FUNCTION_BLOCK FiveStateActuator (* Basic Function Block Type *)
  (* Standard: 61499-2 *)
  (* Version 0.0, 5/13/2025, azam_w, Schneider Electric, Template *)
  PACKAGE Main;
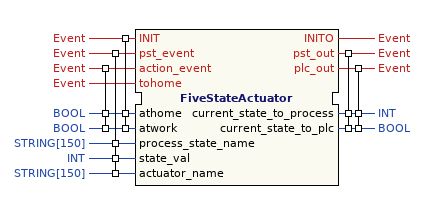
  EVENT_INPUT
    INIT WITH athome, atwork;
    pst_event WITH process_state_name, state_val, actuator_name; (* Normal Execution Request *)
    action_event WITH athome, atwork;
    tohome;
  END_EVENT
  EVENT_OUTPUT
    INITO;
    pst_out WITH current_state_to_process, current_state_to_plc; (* Execution Confirmation *)
    plc_out WITH current_state_to_plc, current_state_to_process;
  END_EVENT
  VAR_INPUT
    athome : BOOL;
    atwork : BOOL;
    process_state_name : STRING[150];
    state_val : INT;
    actuator_name : STRING[150];
  END_VAR
  VAR_OUTPUT
    current_state_to_process : INT; (* Output event qualifier *)
    current_state_to_plc : BOOL;
  END_VAR
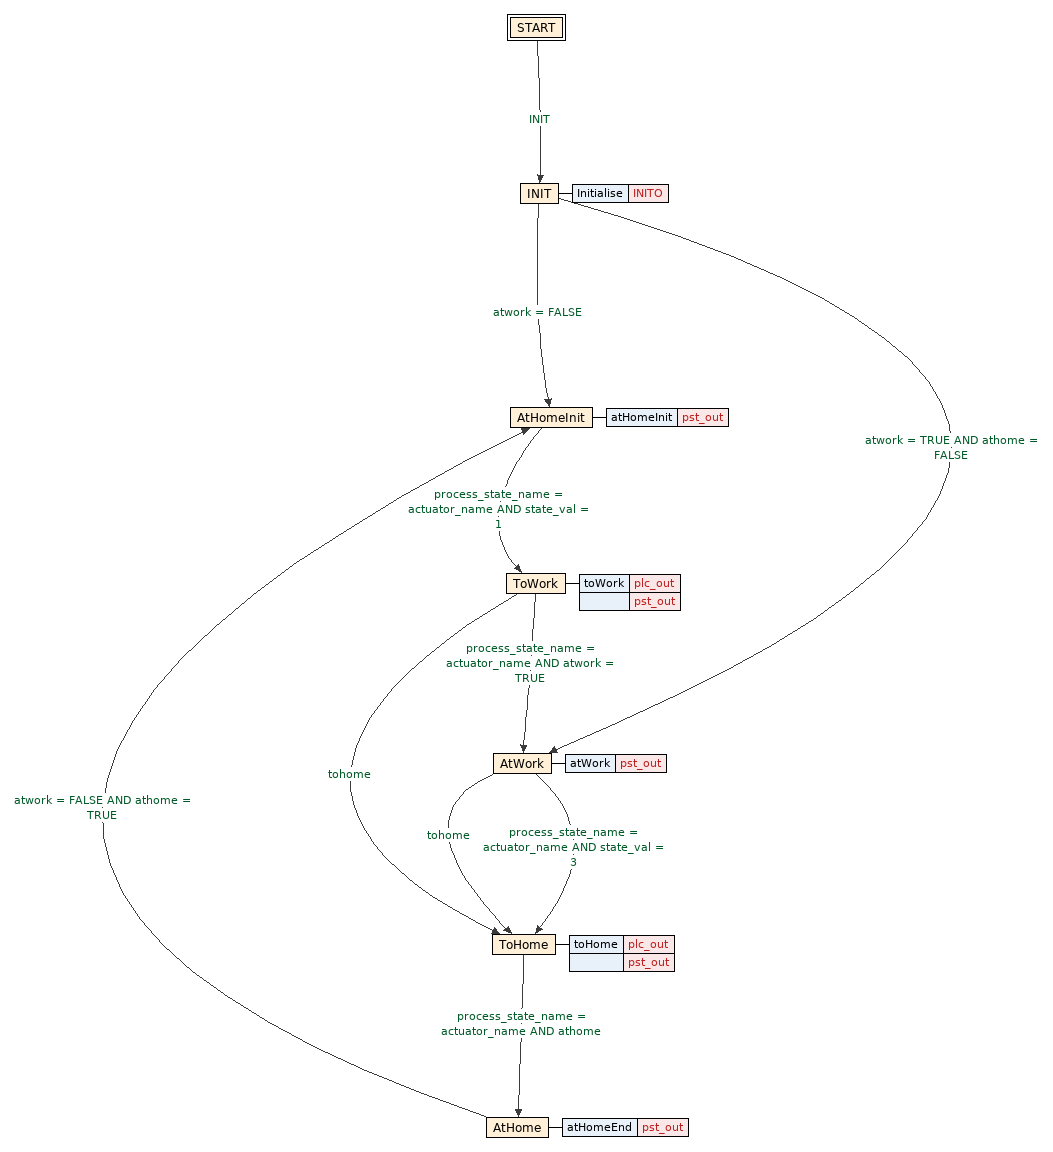
  EC_STATES
    START; (* Initial State *)
    ToWork : toWork -> plc_out, -> pst_out;
    AtWork : atWork -> pst_out;
    ToHome : toHome -> plc_out, -> pst_out;
    AtHome : atHomeEnd -> pst_out;
    AtHomeInit : atHomeInit -> pst_out;
    INIT : Initialise -> INITO;
  END_STATES
  EC_TRANSITIONS
    AtHomeInit TO ToWork := process_state_name = actuator_name AND state_val = 1;
    ToWork TO AtWork := process_state_name = actuator_name AND atwork = TRUE;
    AtHome TO AtHomeInit := atwork = FALSE  AND athome = TRUE;
    ToHome TO AtHome := process_state_name = actuator_name AND athome;
    AtWork TO ToHome := process_state_name = actuator_name AND state_val = 3;
    ToWork TO ToHome := tohome;
    AtWork TO ToHome := tohome;
    START TO INIT := INIT;
    INIT TO AtHomeInit := atwork = FALSE;
    INIT TO AtWork := atwork = TRUE AND athome = FALSE;
  END_TRANSITIONS
  ALGORITHM INIT IN ST: (* Initialization algorithm *)
;
  END_ALGORITHM
  ALGORITHM REQ IN ST: (* Normally executed algorithm *)
;
  END_ALGORITHM
  ALGORITHM toHome IN ST:
;
current_state_to_process := 3;
current_state_to_plc:= FALSE;
  END_ALGORITHM
  ALGORITHM atHomeInit IN ST:
current_state_to_process := 0;
  END_ALGORITHM
  ALGORITHM atWork IN ST:
current_state_to_process := 2;
  END_ALGORITHM
  ALGORITHM toWork IN ST:
;
current_state_to_process := 1;
current_state_to_plc:= TRUE;
  END_ALGORITHM
  ALGORITHM atHomeEnd IN ST:
current_state_to_process := 4;
  END_ALGORITHM
  ALGORITHM Initialise IN ST:
;
  END_ALGORITHM
END_FUNCTION_BLOCK
